// TwinCAT 3 PLC project PLC_modbusFun
// ProgramVersion: 3.1.4024.0
// libraries:
//   PlantControl and CMs, * (ArmAutomation)
//   Tc2_ControllerToolbox, * (Beckhoff Automation GmbH)
//   Tc2_Standard, * (Beckhoff Automation GmbH)
//   Tc2_System, * (Beckhoff Automation GmbH)
//   Tc3_Module, * (Beckhoff Automation GmbH)
// project tree:
//   GVLs/ FIO2.TcGVL, GVL.TcGVL
//   / PlcTask.TcTTO
//   POUs/FBs/ FB_exitConveyorTrigger.TcPOU, FB_exitLoadTrigger.TcPOU, FB_ScaleTrigger.TcPOU, FB_WeightSorter.TcPOU
//   POUs/ FB_ExitSortingConveyors.TcPOU, FB_SortingByWeight.TcPOU, MAIN.TcPOU
// real-time tasks:
//   TASK PlcTask: cycle T#10ms, priority 20, ADS port 350

CONFIGURATION PLC_modbusFun
    RESOURCE PLC ON TwinCAT3
        TASK PlcTask(INTERVAL := T#10ms, PRIORITY := 20);
        PROGRAM MAIN WITH PlcTask : MAIN;
    END_RESOURCE
END_CONFIGURATION

// ---- GVLs/FIO2.TcGVL
{attribute 'qualified_only'}
VAR_GLOBAL
	
	//	Sensor	BOOL	FACTORY I/O (Reset)	498	FALSE
	//	Sensor	Bool	FACTORY I/O (Paused)	497	FALSE
	//	Sensor	Bool	FACTORY I/O (Running)	496	FALSE
	//	Sensor	Bool	Stop	8	TRUE
	//	Sensor	Bool	Start	7	FALSE
	bAtScaleExit : BOOL;	//	Sensor	Bool	At scale exit	2	FALSE
	//	Sensor	Bool	Emergency stop	6	TRUE
	bAtScale : BOOL;	//	Sensor	Bool	At scale	0	FALSE
	bAtExitFront : BOOL;	//	Sensor	Bool	At exit front	5	TRUE
	bAtExitRight : BOOL;//	Sensor	Bool	At exit right	4	TRUE
	bAtExitLeft : BOOL;//	Sensor	Bool	At exit left	3	TRUE
	bAtScaleEntry : BOOL;//	Sensor	Bool	At scale entry	1	TRUE
	//	Sensor	Bool	Reset	9	FALSE
	//	Sensor	Bool	Manual	10	TRUE
	//	Sensor	Bool	Auto	11	FALSE
	bAtLeftEntry : BOOL;	//	Sensor	Bool	At left entry	12	FALSE
	bAtRightEntry : BOOL;//	Sensor	Bool	At right entry	13	FALSE
	bAtForwardEntry : BOOL;//	Sensor	Bool	At forward entry	14	FALSE
	//	Sensor	Float	FACTORY I/O (Time Scale)	240	0
	rWeight : REAL;//	Sensor	Float	Weight	0	0
	//	Actuator	Bool	FACTORY I/O (Reset)	498	FALSE
	//	Actuator	Bool	FACTORY I/O (Pause)	497	FALSE
	//	Actuator	Bool	FACTORY I/O (Run)	496	FALSE
	//	Actuator	Bool	Reset light	15	FALSE
	//	Actuator	Bool	Stop light	14	FALSE
	//	Actuator	Bool	Start light	13	FALSE
	bConveyorLeft : BOOL;	//	Actuator	Bool	Left conveyor	8	FALSE
	bConveyorFront : BOOL;	//	Actuator	Bool	Front conveyor	9	FALSE
	bConveyorRight : BOOL;	//	Actuator	Bool	Right conveyor	7	FALSE
	//	Actuator	Bool	Remover	12	TRUE
	//	Actuator	Bool	Remover	10	TRUE
	//	Actuator	Bool	Remover	11	TRUE
	bSendRight : BOOL;	//	Actuator	Bool	Send right	6	FALSE
	bSendLeft : BOOL;	//	Actuator	Bool	Send left	5	FALSE
	bSendForward : BOOL;	//	Actuator	Bool	Send forward	4	FALSE
	bEmitter : BOOL;	//	Actuator	Bool	Emitter	3	TRUE
	bConveyorEntry : BOOL;//	Actuator	Bool	Entry conveyor	2	FALSE
	bLoadScale : BOOL;//	Actuator	Bool	Load scale	0	FALSE
	//	Actuator	Bool	-	1	FALSE
	//	Actuator	Int	FACTORY I/O (Camera Position)	240	0
	iLeftCount : INT;	//	Actuator	Int	Left count	3	0
	iRightCount : INT;	//	Actuator	Int	Right count	2	0
	iForwardCount : INT;	//	Actuator	Int	Forward count	1	0
	//	Actuator	Int	Weight	0	0

END_VAR

// ---- GVLs/GVL.TcGVL
{attribute 'qualified_only'}
VAR_GLOBAL
	
 mb_Input_Coils    :    ARRAY [0..255] OF BOOL;
 mb_Output_Coils :    ARRAY [0..255] OF BOOL;
 mb_Input_Registers :    ARRAY [0..255] OF WORD; // Modbus TCP master side function code = 04 (read only)
 mb_Output_Registers :    ARRAY [0..255] OF WORD; // Modbus TCP master side function code = 03 & 16 (read/write)
 
 iPackageSize : INT;
 
 smallPackage : BOOL;
 mediumPackage : BOOL;
 largePackage : BOOL;
 
 WeighingDone : BOOL;

END_VAR

// ---- POUs/MAIN.TcPOU
PROGRAM MAIN
VAR
	fbPlant : PlantAndCMs.FB_PlantControl_mode_1;
	udt_plant_data_control : PlantAndCMs.Udt_PlantControl_Mode_1;
	
	fbSortingByWeight : FB_SortingByWeight;
	
	fbExitConveyors : FB_ExitSortingConveyors;
	
	fbScaleTrigger : FB_ScaleTrigger;
	fbExitLoadTrigger : FB_exitLoadTrigger;
	fbExitConveyorTrigger : FB_exitConveyorTrigger;
	
	fbWeightSorter : FB_WeightSorter;
	
	startButton : BOOL;
	
END_VAR

startButton := FALSE;

IF GVL.mb_Output_Coils[1] THEN
	startButton := TRUE;
END_IF

fbPlant(
	Ctrl_Plant := udt_plant_data_control,
	Auto_In := PlantAndCMs.FIO.bAuto,
	 
	Start_In := GVL.mb_Output_Coils[5],
	
	Stop_In := GVL.mb_Output_Coils[6],
	EmgStop_In := PlantAndCMs.FIO.bEmgStop

	);
	
	
fbSortingByWeight(
	control_data := udt_plant_data_control
	);

fbExitConveyors(
	);


fbScaleTrigger(
	scaleEntry_input := FIO2.bAtScaleEntry,
	scaleExit_input := FIO2.bAtScaleExit
		);
		
fbExitLoadTrigger(
	input_left := FIO2.bAtLeftEntry,
	input_right := FIO2.bAtRightEntry,
	input_forward := FIO2.bAtForwardEntry
	
	);
fbExitConveyorTrigger(
	inputLeft := FIO2.bAtExitLeft,
	inputRight := FIO2.bAtExitRight,
	inputForward := FIO2.bAtExitFront,	
	);
	
	
(*fbWeightSorter(
	weight_input := FIO2.rWeight,
	
	small => GVL.smallPackage,
	medium => GVL.mediumPackage,
	large => GVL.largePackage
	
	
	);*)

END_PROGRAM

// ---- POUs/FB_SortingByWeight.TcPOU
FUNCTION_BLOCK FB_SortingByWeight
VAR_INPUT
END_VAR
VAR_OUTPUT
END_VAR
VAR
	WeighingDone : BOOL;
	dummy : BOOL;
END_VAR
VAR_IN_OUT
	control_data : PlantAndCMs.Udt_PlantControl_Mode_1;
	
END_VAR

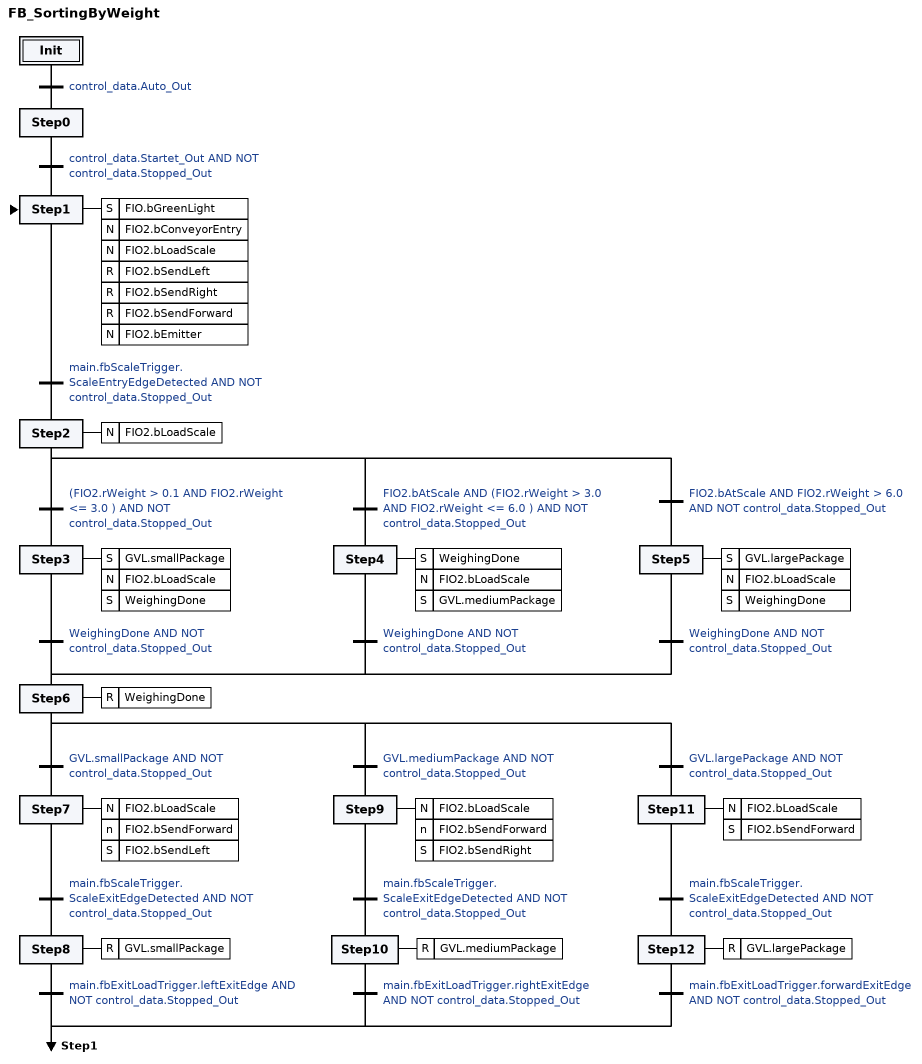
INITIAL_STEP Init:
END_STEP
TRANSITION FROM Init TO Step0
    := control_data.Auto_Out;
END_TRANSITION
STEP Step0:
END_STEP
TRANSITION FROM Step0 TO Step1
    := control_data.Startet_Out AND NOT control_data.Stopped_Out;
END_TRANSITION
STEP Step1:
    FIO.bGreenLight(S);
    FIO2.bConveyorEntry(N);
    FIO2.bLoadScale(N);
    FIO2.bSendLeft(R);
    FIO2.bSendRight(R);
    FIO2.bSendForward(R);
    FIO2.bEmitter(N);
END_STEP
TRANSITION FROM Step1 TO Step2
    := main.fbScaleTrigger.ScaleEntryEdgeDetected AND NOT control_data.Stopped_Out;
END_TRANSITION
STEP Step2:
    FIO2.bLoadScale(N);
END_STEP
TRANSITION FROM Step2 TO Step3
    := (FIO2.rWeight > 0.1 AND FIO2.rWeight <= 3.0 ) AND NOT control_data.Stopped_Out;
END_TRANSITION
STEP Step3:
    GVL.smallPackage(S);
    FIO2.bLoadScale(N);
    WeighingDone(S);
END_STEP
TRANSITION FROM Step3 TO Step6
    := WeighingDone AND NOT control_data.Stopped_Out;
END_TRANSITION
TRANSITION FROM Step2 TO Step4
    := FIO2.bAtScale AND (FIO2.rWeight > 3.0 AND FIO2.rWeight <= 6.0 ) AND NOT control_data.Stopped_Out;
END_TRANSITION
STEP Step4:
    WeighingDone(S);
    FIO2.bLoadScale(N);
    GVL.mediumPackage(S);
END_STEP
TRANSITION FROM Step4 TO Step6
    := WeighingDone AND NOT control_data.Stopped_Out;
END_TRANSITION
TRANSITION FROM Step2 TO Step5
    := FIO2.bAtScale AND FIO2.rWeight > 6.0 AND NOT control_data.Stopped_Out;
END_TRANSITION
STEP Step5:
    GVL.largePackage(S);
    FIO2.bLoadScale(N);
    WeighingDone(S);
END_STEP
TRANSITION FROM Step5 TO Step6
    := WeighingDone AND NOT control_data.Stopped_Out;
END_TRANSITION
STEP Step6:
    WeighingDone(R);
END_STEP
TRANSITION FROM Step6 TO Step7
    := GVL.smallPackage AND NOT control_data.Stopped_Out;
END_TRANSITION
STEP Step7:
    FIO2.bLoadScale(N);
    FIO2.bSendForward(n);
    FIO2.bSendLeft(S);
END_STEP
TRANSITION FROM Step7 TO Step8
    := main.fbScaleTrigger.ScaleExitEdgeDetected AND NOT control_data.Stopped_Out;
END_TRANSITION
STEP Step8:
    GVL.smallPackage(R);
END_STEP
TRANSITION FROM Step8 TO Step1
    := main.fbExitLoadTrigger.leftExitEdge AND NOT control_data.Stopped_Out;
END_TRANSITION
TRANSITION FROM Step6 TO Step9
    := GVL.mediumPackage AND NOT control_data.Stopped_Out;
END_TRANSITION
STEP Step9:
    FIO2.bLoadScale(N);
    FIO2.bSendForward(n);
    FIO2.bSendRight(S);
END_STEP
TRANSITION FROM Step9 TO Step10
    := main.fbScaleTrigger.ScaleExitEdgeDetected AND NOT control_data.Stopped_Out;
END_TRANSITION
STEP Step10:
    GVL.mediumPackage(R);
END_STEP
TRANSITION FROM Step10 TO Step1
    := main.fbExitLoadTrigger.rightExitEdge AND NOT control_data.Stopped_Out;
END_TRANSITION
TRANSITION FROM Step6 TO Step11
    := GVL.largePackage AND NOT control_data.Stopped_Out;
END_TRANSITION
STEP Step11:
    FIO2.bLoadScale(N);
    FIO2.bSendForward(S);
END_STEP
TRANSITION FROM Step11 TO Step12
    := main.fbScaleTrigger.ScaleExitEdgeDetected AND NOT control_data.Stopped_Out;
END_TRANSITION
STEP Step12:
    GVL.largePackage(R);
END_STEP
TRANSITION FROM Step12 TO Step1
    := main.fbExitLoadTrigger.forwardExitEdge AND NOT control_data.Stopped_Out;
END_TRANSITION

END_FUNCTION_BLOCK

// ---- POUs/FB_ExitSortingConveyors.TcPOU
FUNCTION_BLOCK FB_ExitSortingConveyors
VAR_INPUT
	bStop : BOOL;
	bEmgStop : BOOL;
END_VAR
VAR_OUTPUT
END_VAR
VAR
	dummy : BOOL;
	
	CounterLeft : Tc2_Standard.CTU;
	CounterRight : Tc2_Standard.CTU;
	CounterForward : Tc2_Standard.CTU;
END_VAR

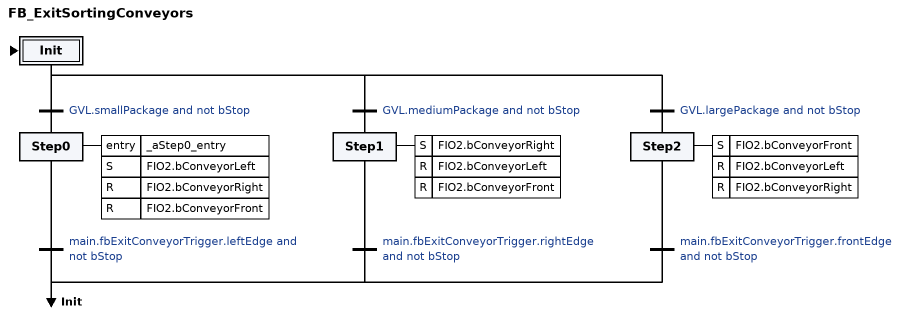
INITIAL_STEP Init:
END_STEP
TRANSITION FROM Init TO Step0
    := GVL.smallPackage and not bStop;
END_TRANSITION
STEP Step0:
    _aStep0_entry(P1);  // entry action
    FIO2.bConveyorLeft(S);
    FIO2.bConveyorRight(R);
    FIO2.bConveyorFront(R);
END_STEP
TRANSITION FROM Step0 TO Init
    := main.fbExitConveyorTrigger.leftEdge and not bStop;
END_TRANSITION
TRANSITION FROM Init TO Step1
    := GVL.mediumPackage and not bStop;
END_TRANSITION
STEP Step1:
    FIO2.bConveyorRight(S);
    FIO2.bConveyorLeft(R);
    FIO2.bConveyorFront(R);
END_STEP
TRANSITION FROM Step1 TO Init
    := main.fbExitConveyorTrigger.rightEdge and not bStop;
END_TRANSITION
TRANSITION FROM Init TO Step2
    := GVL.largePackage and not bStop;
END_TRANSITION
STEP Step2:
    FIO2.bConveyorFront(S);
    FIO2.bConveyorLeft(R);
    FIO2.bConveyorRight(R);
END_STEP
TRANSITION FROM Step2 TO Init
    := main.fbExitConveyorTrigger.frontEdge and not bStop;
END_TRANSITION

END_FUNCTION_BLOCK

// ---- POUs/FBs/FB_ScaleTrigger.TcPOU
FUNCTION_BLOCK FB_ScaleTrigger
VAR_INPUT
	scaleEntry_input : BOOL;
	
	scaleExit_input : BOOL;
END_VAR
VAR_OUTPUT
	ScaleEntryEdgeDetected : BOOL;
	
	ScaleExitEdgeDetected : BOOL;
END_VAR
VAR
	rTrigScaleEntry : Tc2_Standard.R_TRIG;
	
	fTrigScaleExit : Tc2_Standard.F_TRIG;
END_VAR

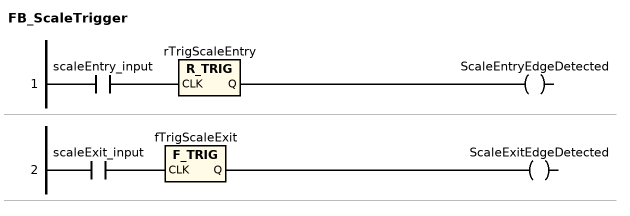
// NETWORK 1
rTrigScaleEntry(CLK := scaleEntry_input); // R_TRIG
ScaleEntryEdgeDetected := rTrigScaleEntry.Q;

// NETWORK 2
fTrigScaleExit(CLK := scaleExit_input); // F_TRIG
ScaleExitEdgeDetected := fTrigScaleExit.Q;

END_FUNCTION_BLOCK

// ---- POUs/FBs/FB_exitLoadTrigger.TcPOU
FUNCTION_BLOCK FB_exitLoadTrigger
VAR_INPUT
	input_right : BOOL;
	input_left : BOOL;
	input_forward : BOOL;
	
END_VAR
VAR_OUTPUT
	leftExitEdge : BOOL;
	rightExitEdge: BOOL;
	forwardExitEdge : BOOL;
END_VAR
VAR
	f_trig_left : Tc2_Standard.F_TRIG;
	f_trig_right : Tc2_Standard.F_TRIG;
	f_trig_forward : Tc2_Standard.F_TRIG;
END_VAR

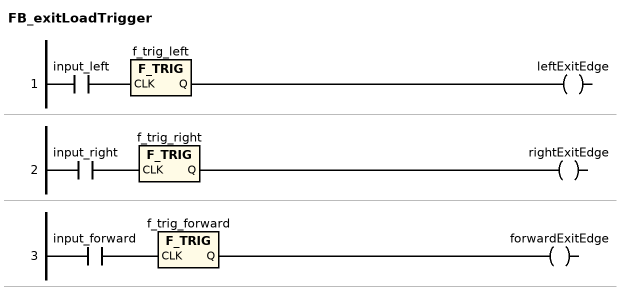
// NETWORK 1
f_trig_left(CLK := input_left); // F_TRIG
leftExitEdge := f_trig_left.Q;

// NETWORK 2
f_trig_right(CLK := input_right); // F_TRIG
rightExitEdge := f_trig_right.Q;

// NETWORK 3
f_trig_forward(CLK := input_forward); // F_TRIG
forwardExitEdge := f_trig_forward.Q;

END_FUNCTION_BLOCK

// ---- POUs/FBs/FB_exitConveyorTrigger.TcPOU
FUNCTION_BLOCK FB_exitConveyorTrigger
VAR_INPUT
	inputLeft : BOOL;
	inputRight : BOOL;
	inputForward : BOOL;
END_VAR
VAR_OUTPUT
	leftEdge : BOOL;
	rightEdge : BOOL;
	frontEdge : BOOL;
END_VAR
VAR
	rTrigLeft : Tc2_Standard.R_TRIG;
	rTrigRight : Tc2_Standard.R_TRIG;
	rTrigForward : Tc2_Standard.R_TRIG;
END_VAR

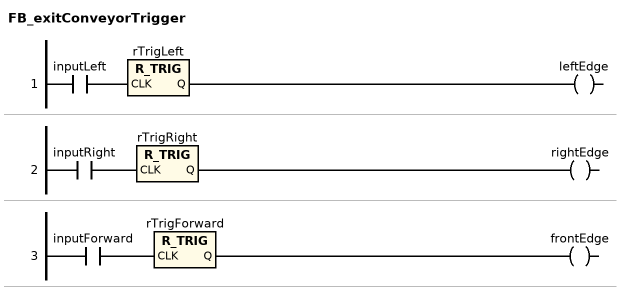
// NETWORK 1
rTrigLeft(CLK := inputLeft); // R_TRIG
leftEdge := rTrigLeft.Q;

// NETWORK 2
rTrigRight(CLK := inputRight); // R_TRIG
rightEdge := rTrigRight.Q;

// NETWORK 3
rTrigForward(CLK := inputForward); // R_TRIG
frontEdge := rTrigForward.Q;

END_FUNCTION_BLOCK

// ---- POUs/FBs/FB_WeightSorter.TcPOU
FUNCTION_BLOCK FB_WeightSorter
VAR_INPUT
	weight_input : REAL;
END_VAR
VAR_OUTPUT
	iPackageSize : INT;
	
	small : BOOL;
	medium : BOOL;
	large : BOOL;
END_VAR
VAR
END_VAR
VAR // added by the converter: edge detectors and wires of the graphical bodies
    _w1, _w2, _w3 : BOOL;
END_VAR

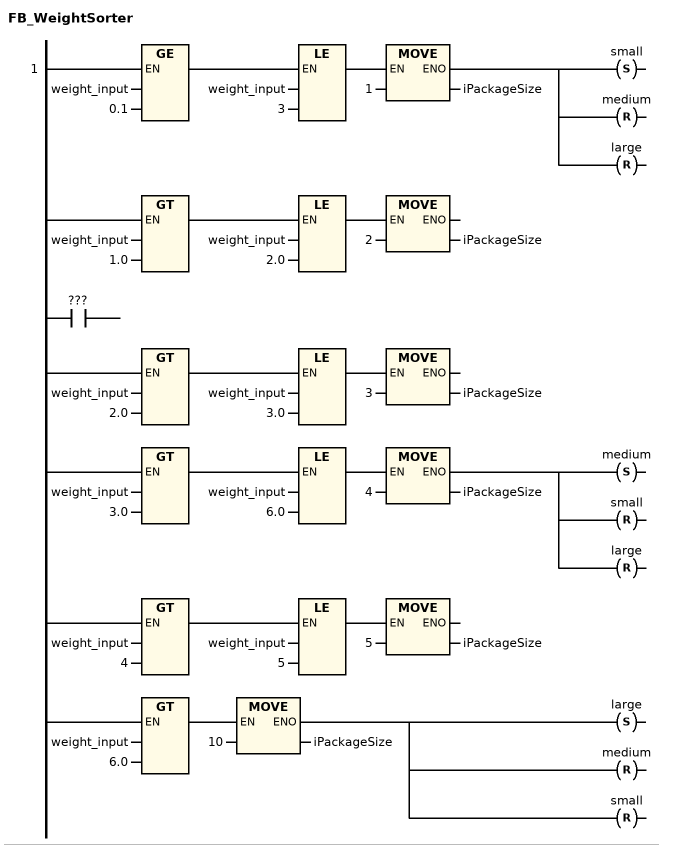
// NETWORK 1
_w1 := weight_input >= 0.1 AND weight_input <= 3;
IF _w1 THEN iPackageSize := 1; END_IF
small S= _w1;
medium R= _w1;
large R= _w1;
IF weight_input > 1.0 AND weight_input <= 2.0 THEN iPackageSize := 2; END_IF
IF weight_input > 2.0 AND weight_input <= 3.0 THEN iPackageSize := 3; END_IF
_w2 := weight_input > 3.0 AND weight_input <= 6.0;
IF _w2 THEN iPackageSize := 4; END_IF
medium S= _w2;
small R= _w2;
large R= _w2;
IF weight_input > 4 AND weight_input <= 5 THEN iPackageSize := 5; END_IF
_w3 := weight_input > 6.0;
IF _w3 THEN iPackageSize := 10; END_IF
large S= _w3;
medium R= _w3;
small R= _w3;

END_FUNCTION_BLOCK
